PROGRAM P70_Interface
VAR
END_VAR

//

END_PROGRAM

(* stored: Version 1.1.0.1, ProductVersion 3.1.4024.15
   POU P70_Interface: Id {9275347a-a4b2-46b6-b185-3a8be1c80031}, SpecialFunc None *)
